(* CODESYS project FU_iBitGetPart.xml

Project tree, tasks and I/O mapping:
  function FU_iBitGetPart [ST]
*)

// FU_iBitGetPart
//This function gets only the needed bits of a variable
// |**Version**|**Author**| **Date** |**Changes**
// | 1         | NSN      | 16-03-22 | Creation
FUNCTION FU_iBitGetPart : INT
VAR_INPUT
	value			:INT;		//Variable to get value from
	amount			:BYTE;		//Amount of bits to change
	offset			:BYTE;		//Offset in variable to change bits at
END_VAR

FU_iBitGetPart		:=		TO_INT(SHR(TO_UINT(value),offset) AND TO_UINT(GConstants.binaryMaskInt[amount]));

END_FUNCTION
